// TIA Portal project "MAT CON INVERTER" (V11)

(* hardware
DEVICE "Stazione SIMATIC 1200_1"  S71200.Device
   slot 0: "Telaio di montaggio S7-1200"  Rack  V1.0
   slot 1: "PLC_1"  CPU 1200 non specificata  6ES7 2XX-XXXX-XXXX  V2.1
*)

// ===== PLC "PLC_1"  CPU 1200 non specificata =====

VAR_GLOBAL   // PLC tag table "Tabella delle variabili standard"
   "STATO" AT %MW0 : Int;
   "PEM" AT %I0.0 : Bool;
   "ON" AT %I0.1 : Bool;
   "STOP" AT %I0.2 : Bool;
   "VERSO SX" AT %I0.3 : Bool;
   "VERSO DX" AT %I0.4 : Bool;
   "ON/OFF" AT %Q0.0 : Bool;
   "VERSO" AT %Q0.1 : Bool;
   "VERSO SX LED" AT %Q0.5 : Bool;
   "VERSO DX LED" AT %Q0.6 : Bool;
   "LED EM" AT %Q0.7 : Bool;
   "LED ALIM" AT %Q1.0 : Bool;
END_VAR

ORGANIZATION_BLOCK "Main"   // OB1, LAD, ProgramCycle
TITLE = "Main Program Sweep (Cycle)"
{ S7_Optimized_Access := 'FALSE' }
VERSION : 0.1
   VAR_TEMP   // added for the SCL form of the ladder/FBD networks
      _w1 : Bool;
   END_VAR
BEGIN

REGION Network 1: STATO INIZIALE/EMERGENZA
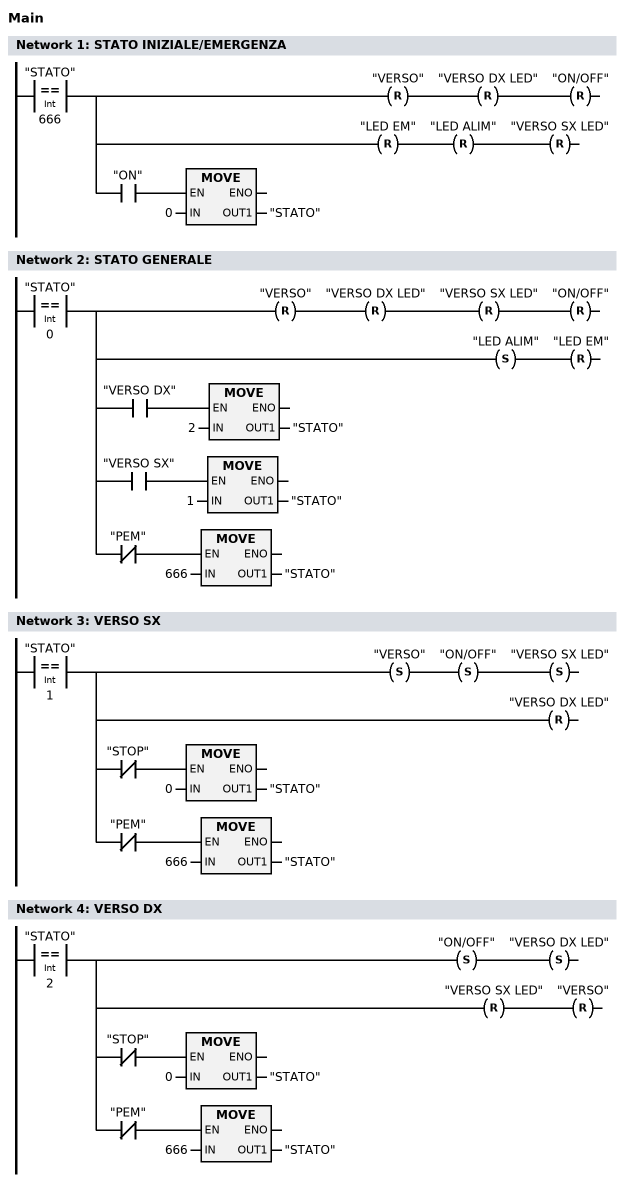
   RUNG wire#powerrail
      { S7_Templates := "SrcType := Int" } EQ_Contact(in1 := "STATO", in2 := 666)
      wire#w1
      R_Coil( "VERSO" )
      R_Coil( "VERSO DX LED" )
      R_Coil( "ON/OFF" )
   END_RUNG
   RUNG wire#w1
      R_Coil( "LED EM" )
      R_Coil( "LED ALIM" )
      R_Coil( "VERSO SX LED" )
   END_RUNG
   RUNG wire#w1
      Contact( "ON" )
      { S7_GenerateENO := "TRUE" } Move(in := 0, out1 => "STATO")
   END_RUNG
   // the same network as SCL:
   #_w1 := "STATO" = 666;
   IF #_w1 THEN
       "VERSO" := FALSE;
       "VERSO DX LED" := FALSE;
       "ON/OFF" := FALSE;
       "LED EM" := FALSE;
       "LED ALIM" := FALSE;
       "VERSO SX LED" := FALSE;
   END_IF;
   IF #_w1 AND "ON" THEN "STATO" := 0; END_IF;
END_REGION

REGION Network 2: STATO GENERALE
   RUNG wire#powerrail
      { S7_Templates := "SrcType := Int" } EQ_Contact(in1 := "STATO", in2 := 0)
      wire#w1
      R_Coil( "VERSO" )
      R_Coil( "VERSO DX LED" )
      R_Coil( "VERSO SX LED" )
      R_Coil( "ON/OFF" )
   END_RUNG
   RUNG wire#w1
      S_Coil( "LED ALIM" )
      R_Coil( "LED EM" )
   END_RUNG
   RUNG wire#w1
      Contact( "VERSO DX" )
      { S7_GenerateENO := "TRUE" } Move(in := 2, out1 => "STATO")
   END_RUNG
   RUNG wire#w1
      Contact( "VERSO SX" )
      { S7_GenerateENO := "TRUE" } Move(in := 1, out1 => "STATO")
   END_RUNG
   RUNG wire#w1
      I_Contact( "PEM" )
      { S7_GenerateENO := "TRUE" } Move(in := 666, out1 => "STATO")
   END_RUNG
   // the same network as SCL:
   #_w1 := "STATO" = 0;
   IF #_w1 THEN
       "VERSO" := FALSE;
       "VERSO DX LED" := FALSE;
       "VERSO SX LED" := FALSE;
       "ON/OFF" := FALSE;
       "LED ALIM" := TRUE;
       "LED EM" := FALSE;
   END_IF;
   IF #_w1 AND "VERSO DX" THEN "STATO" := 2; END_IF;
   IF #_w1 AND "VERSO SX" THEN "STATO" := 1; END_IF;
   IF #_w1 AND NOT "PEM" THEN "STATO" := 666; END_IF;
END_REGION

REGION Network 3: VERSO SX
   RUNG wire#powerrail
      { S7_Templates := "SrcType := Int" } EQ_Contact(in1 := "STATO", in2 := 1)
      wire#w1
      S_Coil( "VERSO" )
      S_Coil( "ON/OFF" )
      S_Coil( "VERSO SX LED" )
   END_RUNG
   RUNG wire#w1
      R_Coil( "VERSO DX LED" )
   END_RUNG
   RUNG wire#w1
      I_Contact( "STOP" )
      { S7_GenerateENO := "TRUE" } Move(in := 0, out1 => "STATO")
   END_RUNG
   RUNG wire#w1
      I_Contact( "PEM" )
      { S7_GenerateENO := "TRUE" } Move(in := 666, out1 => "STATO")
   END_RUNG
   // the same network as SCL:
   #_w1 := "STATO" = 1;
   IF #_w1 THEN
       "VERSO" := TRUE;
       "ON/OFF" := TRUE;
       "VERSO SX LED" := TRUE;
       "VERSO DX LED" := FALSE;
   END_IF;
   IF #_w1 AND NOT "STOP" THEN "STATO" := 0; END_IF;
   IF #_w1 AND NOT "PEM" THEN "STATO" := 666; END_IF;
END_REGION

REGION Network 4: VERSO DX
   RUNG wire#powerrail
      { S7_Templates := "SrcType := Int" } EQ_Contact(in1 := "STATO", in2 := 2)
      wire#w1
      S_Coil( "ON/OFF" )
      S_Coil( "VERSO DX LED" )
   END_RUNG
   RUNG wire#w1
      R_Coil( "VERSO SX LED" )
      R_Coil( "VERSO" )
   END_RUNG
   RUNG wire#w1
      I_Contact( "STOP" )
      { S7_GenerateENO := "TRUE" } Move(in := 0, out1 => "STATO")
   END_RUNG
   RUNG wire#w1
      I_Contact( "PEM" )
      { S7_GenerateENO := "TRUE" } Move(in := 666, out1 => "STATO")
   END_RUNG
   // the same network as SCL:
   #_w1 := "STATO" = 2;
   IF #_w1 THEN
       "ON/OFF" := TRUE;
       "VERSO DX LED" := TRUE;
       "VERSO SX LED" := FALSE;
       "VERSO" := FALSE;
   END_IF;
   IF #_w1 AND NOT "STOP" THEN "STATO" := 0; END_IF;
   IF #_w1 AND NOT "PEM" THEN "STATO" := 666; END_IF;
END_REGION
END_ORGANIZATION_BLOCK

ORGANIZATION_BLOCK "Startup"   // OB100, LAD, Startup
TITLE = "Complete Restart"
{ S7_Optimized_Access := 'FALSE' }
VERSION : 0.1
   VAR_INPUT
      LostRetentive : Bool;   // True if retentive data are lost
      LostRTC : Bool;   // True if real time clock is lost
   END_VAR
BEGIN

REGION Network 1: STARTUP
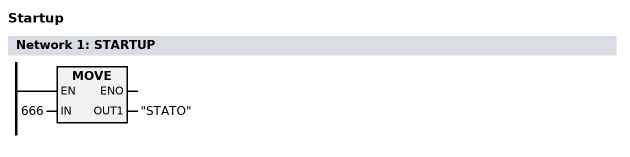
   RUNG wire#powerrail
      { S7_GenerateENO := "TRUE" } Move(in := 666, out1 => "STATO")
   END_RUNG
   // the same network as SCL:
   "STATO" := 666;
END_REGION
END_ORGANIZATION_BLOCK